TYPE U_OdriveRealBytes :
UNION
    Value : REAL;
    Bytes : ARRAY[0..3] OF BYTE;
END_UNION
END_TYPE

(* stored: Version 1.1.0.1
   DUT U_OdriveRealBytes: Id {FBD9E32E-F860-42B3-92F5-A5C692D02503} *)
